// TwinCAT 3 PLC project HelloWorldPlc
// ProgramVersion: 3.1.4023.0
// libraries:
//   Tc2_Standard, * (Beckhoff Automation GmbH)
//   Tc2_System, * (Beckhoff Automation GmbH)
//   Tc3_Module, * (Beckhoff Automation GmbH)
// project tree:
//   / PlcTask.TcTTO
//   POUs/ MAIN.TcPOU

CONFIGURATION HelloWorldPlc
    RESOURCE PLC ON TwinCAT3
        TASK PlcTask(INTERVAL := T#10ms, PRIORITY := 20);
        PROGRAM MAIN WITH PlcTask : MAIN;
    END_RESOURCE
END_CONFIGURATION

// ---- POUs/MAIN.TcPOU
PROGRAM MAIN
VAR
	bRunOnlyOnce : BOOL := TRUE;
	//sHelloWorldStr : STRING := 'Hello World!';
END_VAR

(*Hello World Example - Treat body as an endless while loop therfore a boolean statement is required to keep program from running indefinitely*)

IF bRunOnlyOnce THEN		//boolean statement, IF NOT can be used when bRunOnlyOnce is declared as FALSE
	ADSLOGSTR (
		msgCtrlMask := ADSLOG_MSGTYPE_ERROR, 		//outputs as an error message
		msgFmtStr := 'Hello World',					//'Hello %s' %s points to strArg or sHelloWorldStr
		strArg := '');
	bRunOnlyOnce := FALSE;							//update boolean to false
END_IF

END_PROGRAM
